{attribute 'GeneratedUsingTerminal: ELX3181-0000-0016'}
{attribute addProperty BoxType "ELX3181-0000-0016"}
{attribute addProperty Id "StatusAT %I*Status_05CE4FB58ValueAT %I*INT2"}
{attribute addProperty CRC "1200930947"}
{attribute addProperty Size "10"}
TYPE Ch_1_Al_Inputs_4794C083 :
STRUCT
	{attribute addProperty Name "Status"}
	Status AT %I* : Status_05CE4FB5;
	{attribute addProperty Name "Value"}
	Value AT %I* : INT;
END_STRUCT
END_TYPE

(* stored: Version 1.2.0.0, ProductVersion 3.1.4024.9
   DUT Ch_1_Al_Inputs_4794C083: Id {a8755d60-0508-44dc-a03a-473dfaeb6c29} *)
